{attribute 'qualified_only'}
{attribute 'strict'}
{attribute 'to_string'}
TYPE ST120_Pnp_e :
(
    RESET := 0, // Reset

    INIT := 100, // Initialisieren 
    Init_HomeVerticals,
    Init_VerticalsUp,
    Init_HomeHorizontals,
    Init_HorizontalsToTrack,
    Init_check_if_pces_handled,

    READY := 999,  // READY to Start, Init Done 
    START := 1000, // Start Zyklisch
    MOVER_FREE_OP, // Ab here, operation without mover can be done

    PnP_Hor_ToRotTablePos,
    PnP_WaitOnFeeder,
    PnP_Ver_RotTableDown,
    Gripper_open,
    PnP_Ver_RotTableUp,
    PnP_Hor_ToTrackPos,
    waitOnMover,     // wait until the mover is there
    MOVER_NEEDED_OP, // Since here, a mover in position is needed to perform the action

    PnP_Ver_ShuttleDown,
    PnP_Ver_ShuttleTorqueControl,
    Gripper_close,
    PnP_Ver_ShuttleUp,

    SYNC_MOVER_LEAVE, // MoverMan need to take the mover
    DONE := 8000,     // Ablauf beendet 
    ERROR := 9000,    // Fehler 
    _max
);
END_TYPE

(* stored: Version 1.1.0.1, ProductVersion 3.1.4024.6
   EnumerationTextList ST120_Pnp_e: Id {e5aa6d13-808a-40a0-9bc2-b44aeab332eb} *)
